FUNCTION_BLOCK EM_DockingInterface EXTENDS EM_Base
VAR CONSTANT 
	c_nResultDataSize : UINT := 20;
END_VAR
VAR
//------------------------------------------//
//Control Modules (Devices)
	cmValveDockingClampsUpper : CM_ValveWithDoubleFB;
	cmValveDockingClampsLower : CM_ValveWithDoubleFB;
	cmValveUnlockingPinsUpper : CM_ValveWithFB;
	cmValveUnlockingPinsLower : CM_ValveWithFB;
	
//------------------------------------------//

//------------------------------------------//
//Inputs
		s_diStaBoxAtPreDockingPosition : FB_DigInput;
		s_diStaSensorBoxAtDockedPosition : FB_DigInput;
		
//------------------------------------------//
	
//------------------------------------------//
//Outputs

//------------------------------------------//


//Requests
	s_bReqDockBox : BOOL := FALSE;
	s_bReqUndockBox : BOOL := FALSE;
	
//Properties
	s_bStaDockingDone : BOOL := FALSE;
	s_bStaUndockingDone : BOOL := FALSE;
	
	
//Alarms

//Warnings
	fbAlarmHandlerNoBoxPresentAtPreDockingPosition : FB_AlarmHandler;
	fbAlarmHandlerNoBoxPresentAtDockedPosition : FB_AlarmHandler;

	s_bWrnNoBoxPresentAtPreDockingPosition : BOOL;
	s_bWrnNoBoxPresentAtDockedPosition : BOOL;
	
//------------------------------------------//
//Params
	//Tool settings
	s_fbParamToolHardwareNr				: FB_HmiParamHandler;
    s_fbParamToolSoftwareVersion		: FB_HmiParamHandler;

	s_fbParamName						: FB_HmiParamHandler;
	s_fbParamNumber						: FB_HmiParamHandler;
	s_fbParamRevision                   : FB_HmiParamHandler;
	
	s_fbParamTeslaMeterIp				: FB_HmiParamHandler;
	s_fbParamTeslaMeterPort				: FB_HmiParamHandler;
	
	//Product settings (Maybe)
	s_fbParamTotalStroke				: FB_HmiParamHandler;
	s_fbParamStepStroke					: FB_HmiParamHandler;
	s_fbParamAveragingNumberTest		: FB_HmiParamHandler;
	
	s_fbParamaMaxMagnitudeCriteria		: FB_HmiParamHandler;
	
	s_fbParamRefIduBottom				: FB_HmiParamHandler;
	s_fbParamRefItm                     : FB_HmiParamHandler;
	s_fbParamRefCenterTpmPipe           : FB_HmiParamHandler;
	s_fbParamRefCpValve					: FB_HmiParamHandler;
//------------------------------------------//

//------------------------------------------//
//Variables
	s_sTestResult 						: STRING;
	
	s_eSeqDockingInterface : E_SeqDockingInterface;
	s_fbSeqDockingInterface : FB_SeqControl;
	
	s_eCurrentTest						: E_TestMode;
//--	s_stCommandsTesla					: ST_SCPI_TeslaCommands;
	
	
	// Interlocks
	s_bIlckSpeedDoorOuterToOpen 		: BOOL := TRUE;
	s_bIlckSpeedDoorOuterToClose 		: BOOL := TRUE;
	
	s_bIlckDoorLockCleanroomToOpen 		: BOOL := TRUE;
	
//------------------------------------------//

//------------------------------------------//
//Sensor data	
	s_aMagneticX						: ARRAY[0..c_nResultDataSize] OF LREAL;
	s_aMagneticY						: ARRAY[0..c_nResultDataSize] OF LREAL;
	s_aMagneticZ						: ARRAY[0..c_nResultDataSize] OF LREAL;
	s_aMagneticMagnitude				: ARRAY[0..c_nResultDataSize] OF LREAL;
	s_aProbePositionZ					: ARRAY[0..c_nResultDataSize] OF LREAL;
	
	s_sXMLData							: STRING(Param_Project.n_MaxLenghtXmlDbRow*Param_Project.n_NumberofRowsXmlDb);
	
	s_aHmi_MagneticTest					: ARRAY[1..3,0..c_nResultDataSize] OF ST_POINT;
	
//	s_aHmi_ProbePositionZ				: ARRAY[1..1,1..GVL_Datalogging.c_nHmiLogSize] OF ST_POINT;
//------------------------------------------//

//------------------------------------------//
//Alarms

//------------------------------------------//

//------------------------------------------//
//Hmi
	s_nToHmiStepNr						: INT;
	s_nToHmiMaxStepNr					: INT;
	s_sToHmiInstructionText				: T_MAXSTRING;
	s_sToHmiProcedure					: T_MAXSTRING;
	
	s_fbHmiBtnStart						: FB_HmiBtn;
	s_fbHmiBtnStop						: FB_HmiBtn;	
	s_fbHmiBtnDiagnosticsLogging		: FB_HmiBtn;
	
	s_fbHmiProbeMotor 					: Hmi_Motor_Base;
	
	s_fbHmiBtnEnableMotor				: FB_HmiBtn;
	s_fbHmiBtnHomeMotor					: FB_HmiBtn;
	s_fbHmiBtnGetField					: FB_HmiBtn;
	
	s_fbHmiLedHomedMotor				: FB_HmiLed;
	s_fbHmiTableDownPressed				: FB_HmiLed;
	s_fbHmiStopPressed					: FB_HmiLed;
	s_fbHmiTableDownSensor				: FB_HmiLed;
//------------------------------------------//
END_VAR


SUPER^();

METHOD PROTECTED _m_Alarms : BOOL





IF NOT SUPER^._m_Alarms() THEN
	RETURN;
END_IF

// Set error bits

// Alarm Handlers
fbAlarmHandlerNoBoxPresentAtPreDockingPosition(
	i_bStaActive := s_bWrnNoBoxPresentAtPreDockingPosition, 
	i_eAlarmLevel := E_AlarmLevel.Warning, 
	i_sAlarmText := 'No box present at per-docking position');
	
fbAlarmHandlerNoBoxPresentAtDockedPosition(
	i_bStaActive := s_bWrnNoBoxPresentAtDockedPosition, 
	i_eAlarmLevel := E_AlarmLevel.Warning, 
	i_sAlarmText := 'No box present at docked position');

// Reset warnings
IF i_bCmdReset THEN
	s_bWrnNoBoxPresentAtPreDockingPosition := FALSE;
	s_bWrnNoBoxPresentAtDockedPosition := FALSE;
END_IF	
	
_m_Alarms := TRUE;
END_METHOD

METHOD PROTECTED _m_Devices : BOOL

IF NOT SUPER^._m_Devices() THEN
	RETURN;
END_IF


s_diStaBoxAtPreDockingPosition(
	i_stSettings := );

s_diStaSensorBoxAtDockedPosition(
	i_stSettings := );

cmValveDockingClampsUpper(
	i_bReqEnable := i_bReqEnable,
	i_eCtrlMode := i_eCtrlMode,
	i_bCmdReset := i_bCmdReset,
	i_sCmName := 'Docking clamps upper', 
	i_stSettings := );
	
cmValveDockingClampsLower(
	i_bReqEnable := i_bReqEnable,
	i_eCtrlMode := i_eCtrlMode,
	i_bCmdReset := i_bCmdReset,
	i_sCmName := 'Docking clamps lower',
	i_stSettings := );
	
cmValveUnlockingPinsUpper(
	i_bReqEnable := i_bReqEnable,
	i_eCtrlMode := i_eCtrlMode,
	i_bCmdReset := i_bCmdReset,
	i_sCmName := 'Unloacking pins upper',
	i_stSettings := );
	
cmValveUnlockingPinsLower(
	i_bReqEnable := i_bReqEnable,
	i_eCtrlMode := i_eCtrlMode,
	i_bCmdReset := i_bCmdReset,
	i_sCmName := 'Unloacking pins lower',
	i_stSettings := );
	
(*	
	// Interlocks (doors must work as an airlock, only one door may be opened at all times)
	s_bIlckSpeedDoorOuterToOpen :=
		s_cmDoorLockCleanroom.p_bStaError
		OR NOT(s_cmDoorLockCleanroom.p_bStaEnabled)
		NOT(s_cmDoorLockCleanroom.p_bStaDoorIsClosed)
		OR NOT (s_cmDoorLockCleanroom.p_bStaLockIsApplied)
		OR s_cmDoorLockCleanroom.p_bStaLockIsReleased
		OR TRUE (*Air treathment unit must be running and ok*)
		OR TRUE (*Add more..*);
	s_bIlckSpeedDoorOuterToClose :=
		TRUE (*Opening must be free*)
		OR TRUE (*Add more..*);
	
	s_bIlckDoorLockCleanroomToOpen :=
		s_cmSpeedDoorOuter.p_bStaError
		OR NOT(s_cmSpeedDoorOuter.p_bStaEnabled)
		OR NOT(s_cmSpeedDoorOuter.p_bStaIsClosed)
		OR s_cmSpeedDoorOuter.p_bStaIsClosing
		OR s_cmSpeedDoorOuter.p_bStaIsOpened
		OR s_cmSpeedDoorOuter.p_bStaIsOpening
		OR TRUE (*Air treathment unit must be running and ok*)
		OR TRUE (*Add more..*);
*)	
_m_Devices := TRUE;
END_METHOD

METHOD PROTECTED _m_Hmi : BOOL

IF NOT SUPER^._m_Hmi() THEN
	RETURN;
END_IF

s_fbHmiBtnDiagnosticsLogging();
s_fbHmiBtnStart();
s_fbHmiBtnStop();

s_fbHmiBtnEnableMotor();
s_fbHmiBtnHomeMotor();
s_fbHmiBtnGetField();

s_fbHmiProbeMotor(i_IMotor := s_CmProbeMotor);

s_fbHmiLedHomedMotor(i_bStaLed := s_CmProbeMotor.p_bStaMotorHomed);
s_fbHmiTableDownPressed(i_bStaLed := s_diBtnTableDown.p_bStaInput);
s_fbHmiTableDownSensor(i_bStaLed := s_diTableDownSensor.p_bStaInput);
s_fbHmiStopPressed(i_bStaLed := s_diBtnStop.p_bStaInput);

_m_Hmi := TRUE;
END_METHOD

METHOD PROTECTED _m_Init : BOOL

IF NOT SUPER^._m_Init() THEN
	RETURN;
END_IF

//----------------------------------//
//CM
	s_cmSpeedDoorOuter.i_stSettings.

	s_CmProbeMotor.i_bReqEnable						:= FALSE;
	s_CmProbeMotor.i_sCmName 						:= 'Probe motor';
	s_CmProbeMotor.i_eBtnCtrlType					:= E_HmiButtonType.PUSHBUTTON;
	s_CmProbeMotor.i_bCfgReverseDirection			:= FALSE;
	s_CmProbeMotor.p_bCfgMovingForward				:= TRUE;
	s_CmProbeMotor.p_bCfgMovingReverse				:= TRUE;
	s_CmProbeMotor.p_fSetMotorVelo					:= 10;
	
	s_CmProbeMotor.i_stSettings.i_fAccelaration 	:= 1000;
	s_CmProbeMotor.i_stSettings.i_fDecelaration		:= 1000;
	s_CmProbeMotor.i_stSettings.i_fJerk				:= 10000;
	
	s_CmTeslaMeter.i_bReqEnable						:= FALSE;
	s_CmTeslaMeter.i_stSettings.tConnectionTimeOut	:= T#5S;

	
//---------------------------------//	
	
//----------------------------------//	
//Hmi 
	s_fbHmiBtnDiagnosticsLogging.p_eButtontype 			:= E_HmiButtonType.TOGGLEBUTTON;
	s_fbHmiBtnDiagnosticsLogging.p_bStaVisible 			:= TRUE;
	s_fbHmiBtnDiagnosticsLogging.p_bStaEnabled 			:= TRUE;
	s_fbHmiBtnDiagnosticsLogging.p_sBtnText				:= 'Diagnostics Logging';
	
	s_fbHmiBtnStart.p_eButtontype 						:= E_HmiButtonType.PUSHBUTTON;
	s_fbHmiBtnStart.p_bStaVisible 						:= FALSE;
	s_fbHmiBtnStart.p_bStaEnabled 						:= FALSE;		
	s_fbHmiBtnStart.p_sBtnText							:= 'Start';

	s_fbHmiBtnStop.p_eButtontype 						:= E_HmiButtonType.PUSHBUTTON;
	s_fbHmiBtnStop.p_bStaVisible 						:= FALSE;
	s_fbHmiBtnStop.p_bStaEnabled 						:= FALSE;		
	s_fbHmiBtnStop.p_sBtnText							:= 'Stop';
	
	s_fbHmiBtnEnableMotor.p_eButtontype 				:= E_HmiButtonType.TOGGLEBUTTON;
	s_fbHmiBtnEnableMotor.p_bStaVisible 				:= TRUE;
	s_fbHmiBtnEnableMotor.p_bStaEnabled 				:= FALSE;		
	s_fbHmiBtnEnableMotor.p_sBtnText					:= 'Enable motor';
	
	s_fbHmiBtnGetField.p_eButtontype 					:= E_HmiButtonType.PUSHBUTTON;
	s_fbHmiBtnGetField.p_bStaVisible 					:= TRUE;
	s_fbHmiBtnGetField.p_bStaEnabled 					:= FALSE;		
	s_fbHmiBtnGetField.p_sBtnText						:= 'Get magnetic field';
	
	s_fbHmiBtnHomeMotor.p_eButtontype 					:= E_HmiButtonType.PUSHBUTTON;
	s_fbHmiBtnHomeMotor.p_bStaVisible 					:= TRUE;
	s_fbHmiBtnHomeMotor.p_bStaEnabled 					:= FALSE;		
	s_fbHmiBtnHomeMotor.p_sBtnText						:= 'Home motor';
//----------------------------------//	


//----------------------------------//	
//Initialize all moving averages

//----------------------------------//	

//----------------------------------//	
//Inputs
s_diTableDownSensor.i_stSettings.tmInputDelay	:= T#0S;	
s_diBtnTableDown.i_stSettings.tmInputDelay		:= T#0S;
s_diBtnStop.i_stSettings.tmInputDelay			:= T#0S;
//----------------------------------//	

//----------------------------------//	
//Inputs
s_doRelayTableDown.i_stSettings.bCfgDelay		:= FALSE;	
s_doRelayTableDown.i_stSettings.tmOutputDelay	:= T#0S;	
//----------------------------------//	

_m_Init := TRUE;
END_METHOD

METHOD PROTECTED _m_Inputs : BOOL

IF NOT SUPER^._m_Inputs() THEN
	RETURN;
END_IF

s_diStaBoxAtPreDockingPosition();
s_diStaSensorBoxAtDockedPosition();

_m_Inputs := TRUE;
END_METHOD

METHOD PROTECTED _m_Outputs : BOOL

IF NOT SUPER^._m_Outputs() THEN
	RETURN;
END_IF

s_doRelayTableDown(); //i_bStaOutput written in procedure or manual mode

_m_Outputs := TRUE;
END_METHOD

METHOD PROTECTED _m_Params : BOOL
VAR_INST
	s_fToHmiXAxisMin	: LREAL;
	s_fToHmiXAxisMax	: LREAL;
	s_fToHmiYAxisMin	: LREAL;
	s_fToHmiYAxisMax	: LREAL;
END_VAR

IF NOT SUPER^._m_Params() THEN
	RETURN;
END_IF

s_fbParamToolHardwareNr(i_fDefaultValue				:= 0,
						i_nArrayFolderIndex			:= 1,
						i_sName						:= 'Harware ID',
						i_bIsNumber					:= FALSE);

s_fbParamToolSoftwareVersion(i_fDefaultValue		:= 0,
							i_nArrayFolderIndex		:= 1,
							i_sName					:= 'Software Version',
							i_bIsNumber				:= FALSE);

s_fbParamName(i_fDefaultValue						:= 0,
				i_nArrayFolderIndex					:= 1,
				i_sName								:= 'Description',
				i_bIsNumber							:= FALSE);
							
s_fbParamTeslaMeterIp(i_fDefaultValue			:= 0,
						i_nArrayFolderIndex		:= 1,
						i_sName					:= 'Tesla meter ip adress',
						i_bIsNumber				:= FALSE);
						
s_fbParamTeslaMeterPort(i_fDefaultValue			:= 0,
						i_nArrayFolderIndex		:= 1,
						i_sName					:= 'Tesla meter port number',
						i_bIsNumber				:= TRUE);

//---------

						
s_fbParamTotalStroke(i_fDefaultValue			:= 100,
						i_nArrayFolderIndex		:= 2,
						i_sName					:= 'Total measurement stroke',
						i_bIsNumber				:= TRUE);
						
s_fbParamStepStroke(i_fDefaultValue				:= 10,
						i_nArrayFolderIndex		:= 2,
						i_sName					:= 'Step distance per measurement',
						i_bIsNumber				:= TRUE);

s_fbParamAveragingNumberTest(i_fDefaultValue		:= 10,
							i_nArrayFolderIndex		:= 2,
							i_sName					:= 'Number of measurements per step for averaging the magnetic field',
							i_bIsNumber				:= TRUE);
							
s_fbParamaMaxMagnitudeCriteria(i_fDefaultValue		:= 100,
							i_nArrayFolderIndex		:= 2,
							i_sName					:= 'Maximum allowed magnitude magnetic field (Test)',
							i_bIsNumber				:= TRUE);

s_fbParamRefIduBottom(i_fDefaultValue				:= 0,
							i_nArrayFolderIndex		:= 2,
							i_sName					:= 'Distance from home position to lower IDU Bottom',
							i_bIsNumber				:= TRUE);
							
s_fbParamRefItm(i_fDefaultValue						:= 0,
							i_nArrayFolderIndex		:= 2,
							i_sName					:= 'Distance from home position Itm lower IDU / upper IDU',
							i_bIsNumber				:= TRUE);
							
s_fbParamRefCenterTpmPipe(i_fDefaultValue			:= 0,
							i_nArrayFolderIndex		:= 2,
							i_sName					:= 'Distance from home position to centre TPM pipe',
							i_bIsNumber				:= TRUE);
							
s_fbParamRefCpValve(i_fDefaultValue		:= 0,
							i_nArrayFolderIndex		:= 2,
							i_sName					:= 'Distance from home position to bottom C/P valve',
							i_bIsNumber				:= TRUE);				

GVL_DataLogging.g_stReportData.CabinetSerialNumber      := s_fbParamToolHardwareNr.p_sValue;
GVL_DataLogging.g_stReportData.TesterSoftwareVersion    := s_fbParamToolSoftwareVersion.p_sValue;
GVL_DataLogging.g_stReportData.Operator                 := GVL.g_sUser;
GVL_DataLogging.g_stReportData.Note						:= GVL.g_sNotesEntry;
//GVL_DataLogging.g_stReportData.Message can be filled in test procedure with for example the error if test is stopped
GVL_DataLogging.g_stReportData.SerialNumber             := GVL.g_sSerialNumber;

s_fToHmiXAxisMin	:= -2*s_fbParamaMaxMagnitudeCriteria.p_fValue;
s_fToHmiXAxisMax	:= 2*s_fbParamaMaxMagnitudeCriteria.p_fValue;
s_fToHmiYAxisMin	:= s_CmProbeMotor.p_fHomePosition;
s_fToHmiYAxisMax	:= s_fbParamRefCpValve.p_fValue*1.2;

_m_Params := TRUE;
END_METHOD

METHOD PUBLIC m_DockBox : BOOL

s_bReqDockBox := TRUE;
s_bReqUndockBox := FALSE;

m_DockBox := TRUE;
END_METHOD

METHOD PUBLIC m_Main : BOOL

IF NOT SUPER^.m_Main() THEN
	RETURN;
END_IF


CASE i_eCtrlMode OF

	E_CtrlMode.IDLE:
		;
		
	E_CtrlMode.AUTOMATIC:
		
		s_fbSeqDockingInterface(
			i_nSeqStep := s_eSeqDockingInterface, 
			i_sStepName := , 
			i_bCmdReset := i_bCmdReset, 
			i_bStaError := s_bStaError, 
			q_bStaEntry => , 
			q_tmStepTime => , 
			q_eActState => );
	
		CASE s_eSeqDockingInterface OF
			
			E_SeqDockingInterface.IDLE:
			
				IF s_bReqDockBox THEN
					IF s_diStaBoxAtPreDockingPosition.p_bStaInputDelayed THEN
						s_eSeqDockingInterface := E_SeqDockingInterface.DOCKING_CLOSE_CLAMPS;
					ELSE
						s_bWrnNoBoxPresentAtPreDockingPosition := TRUE;	
					END_IF
				END_IF
				
				IF s_bReqUndockBox THEN
					IF s_diStaSensorBoxAtDockedPosition.p_bStaInputDelayed THEN
						s_eSeqDockingInterface := E_SeqDockingInterface.UNDOCKING_LOCK_DOOR;
					ELSE
						s_bWrnNoBoxPresentAtDockedPosition := TRUE;	
					END_IF	
					
				END_IF
			
				IF s_bReqDockBox AND s_diStaBoxAtPreDockingPosition.p_bStaInputDelayed THEN
					s_eSeqDockingInterface := E_SeqDockingInterface.DOCKING_CLOSE_CLAMPS; 
				ELSIF s_bReqUndockBox THEN	
					s_eSeqDockingInterface := E_SeqDockingInterface.UNDOCKING_LOCK_DOOR;
				END_IF
				
			E_SeqDockingInterface.DOCKING_CLOSE_CLAMPS:
				
				IF s_fbSeqDockingInterface.q_bStaEntry THEN 
					cmValveDockingClampsUpper.m_On();
					cmValveDockingClampsLower.m_On();
				END_IF
				
				IF cmValveDockingClampsUpper.p_bStaIsOn AND cmValveDockingClampsLower.p_bStaIsOn THEN
					s_eSeqDockingInterface := E_SeqDockingInterface.DOCKING_UNLOCK_DOOR;
				ELSIF cmValveDockingClampsUpper.p_bStaError OR cmValveDockingClampsLower.p_bStaError THEN 
					s_eSeqDockingInterface := E_SeqDockingInterface.ERROR;
					// write down some info?
				ELSIF s_fbSeqDockingInterface.q_tmStepTime >= T#30S THEN
 					s_eSeqDockingInterface := E_SeqDockingInterface.ERROR;
					// write down some info?
				END_IF
			
			E_SeqDockingInterface.DOCKING_UNLOCK_DOOR:
			
				IF s_fbSeqDockingInterface.q_bStaEntry THEN 
					cmValveUnlockingPinsUpper.m_On();
					cmValveUnlockingPinsLower.m_On();
				END_IF
				
				IF cmValveUnlockingPinsUpper.p_bStaIsOn AND cmValveUnlockingPinsLower.p_bStaIsOn THEN
					s_eSeqDockingInterface := E_SeqDockingInterface.DOCKING_DONE;
				ELSIF cmValveUnlockingPinsUpper.p_bStaError OR cmValveUnlockingPinsLower.p_bStaError THEN 
					s_eSeqDockingInterface := E_SeqDockingInterface.ERROR;
					// write down some info?
				ELSIF s_fbSeqDockingInterface.q_tmStepTime >= T#30S THEN
 					s_eSeqDockingInterface := E_SeqDockingInterface.ERROR;
					// write down some info?
				END_IF
			
			E_SeqDockingInterface.DOCKING_DONE:
				s_eSeqDockingInterface := E_SeqDockingInterface.IDLE;
			
			E_SeqDockingInterface.UNDOCKING_LOCK_DOOR:
			
				IF s_fbSeqDockingInterface.q_bStaEntry THEN 
					cmValveUnlockingPinsUpper.m_Off();
					cmValveUnlockingPinsLower.m_Off();
				END_IF
				
				IF cmValveUnlockingPinsUpper.p_bStaIsOff AND cmValveUnlockingPinsLower.p_bStaIsOff THEN
					s_eSeqDockingInterface := E_SeqDockingInterface.UNDOCKING_OPEN_CLAMPS;
				ELSIF cmValveUnlockingPinsUpper.p_bStaError OR cmValveUnlockingPinsLower.p_bStaError THEN 
					s_eSeqDockingInterface := E_SeqDockingInterface.ERROR;
					// write down some info?
				ELSIF s_fbSeqDockingInterface.q_tmStepTime >= T#30S THEN
 					s_eSeqDockingInterface := E_SeqDockingInterface.ERROR;
					// write down some info?
				END_IF
				
			E_SeqDockingInterface.UNDOCKING_OPEN_CLAMPS:
			
				IF s_fbSeqDockingInterface.q_bStaEntry THEN 
					cmValveDockingClampsUpper.m_Off();
					cmValveDockingClampsLower.m_Off();
				END_IF
				
				IF cmValveDockingClampsUpper.p_bStaIsOff AND cmValveDockingClampsLower.p_bStaIsOff THEN
					s_eSeqDockingInterface := E_SeqDockingInterface.UNDOCKING_DONE;
				ELSIF cmValveDockingClampsUpper.p_bStaError OR cmValveDockingClampsLower.p_bStaError THEN 
					s_eSeqDockingInterface := E_SeqDockingInterface.ERROR;
					// write down some info?
				ELSIF s_fbSeqDockingInterface.q_tmStepTime >= T#30S THEN
 					s_eSeqDockingInterface := E_SeqDockingInterface.ERROR;
					// write down some info?
				END_IF
				
			E_SeqDockingInterface.UNDOCKING_DONE:
				s_eSeqDockingInterface := E_SeqDockingInterface.IDLE;
				
			E_SeqDockingInterface.READY:
				;
			
			E_SeqDockingInterface.ERROR:
				
				IF i_bCmdReset THEN
					//Reset errors (probebly alredy done in the methode devices)
					//--cmValveDockingClampsUpper.i_bCmdReset := TRUE;
				
					s_eSeqDockingInterface := E_SeqDockingInterface.IDLE;
				END_IF
				
		END_CASE		
	
		
	E_CtrlMode.MANUAL:
		;
	

END_CASE

//-- Old code as an example
(*
CASE i_eCtrlMode OF
	E_CtrlMode.IDLE:
		IF s_CmProbeMotor.p_bStaEnabled THEN
			s_CmProbeMotor.m_DisableAxis();
			s_fbHmiBtnEnableMotor.m_Off();
			s_fbHmiBtnHomeMotor.p_bStaEnabled := FALSE;
		END_IF
		
		s_eCurrentTest	:= 	E_TestMode.IDLE;
	
		s_fbHmiBtnStop.p_bStaVisible := FALSE;
		s_fbHmiBtnStop.p_bStaEnabled := FALSE;		
		
	E_CtrlMode.AUTOMATIC:
		
		CASE s_eCurrentTest OF
			E_TestMode.IDLE:
				GVL.g_bLedFlashSlow			:= FALSE;
				
				s_CmProbeMotor.i_bReqEnable	:= FALSE;
			
				GVL_KMWEGenericLib.g_fbHmiBtnReturn.p_bStaEnabled 	:= TRUE;
				GVL_KMWEGenericLib.g_fbHmiBtnReturn.p_bStaVisible 	:= TRUE;
				
				IF GVL.g_sToHmiMiddleContent = GVL.g_stHmiMiddle.OperatorInputData THEN
					IF NOT GVL_KMWEGenericLib.g_fbAlarmManager.p_bAlarmActive THEN
						s_fbHmiBtnStart.p_bStaVisible	:= TRUE;
						s_fbHmiBtnStart.p_bStaEnabled	:= TRUE;
					ELSE
						s_fbHmiBtnStart.p_bStaVisible	:= FALSE;
						s_fbHmiBtnStart.p_bStaEnabled	:= FALSE;
					END_IF
				END_IF
				
				IF s_fbHmiBtnStart.p_osrBtnPress THEN
					s_eCurrentTest := E_TestMode.Magnetic; 
				END_IF 
				
			E_TestMode.Magnetic:	
				_m_Procedure_Test(i_bCmdReset			:= s_fbHmiBtnStart.p_osfBtnPress, 
									i_bStaError			:= GVL_KMWEGenericLib.g_fbAlarmManager.p_bAlarmActive OR s_fbHmiBtnStop.p_osrBtnPress OR s_diBtnStop.p_osrOn);
		END_CASE
		
	E_CtrlMode.MANUAL:
		_m_Manual(i_bCmdReset			:= GVL.g_UnRMMT.s_fbHmiBtnManual.p_osfBtnPress OR GVL_KMWEGenericLib.g_fbAlarmManager.p_osrReset, 
					i_bStaError			:= GVL_KMWEGenericLib.g_fbAlarmManager.p_bAlarmActive OR s_fbHmiBtnStop.p_osrBtnPress OR s_diBtnStop.p_osrOn);	
END_CASE
*)
END_METHOD

METHOD PUBLIC m_UndockBox : BOOL






s_bReqDockBox := FALSE;
s_bReqUndockBox := TRUE;

m_UndockBox := TRUE;
END_METHOD

PROPERTY PUBLIC p_bStaDockingDone : BOOL
GET

p_bStaDockingDone := s_bStaDockingDone;
END_GET
END_PROPERTY

PROPERTY p_bStaUndockingDone : BOOL
GET

p_bStaUndockingDone := s_bStaUndockingDone;
END_GET
END_PROPERTY

END_FUNCTION_BLOCK

(* stored: Version 1.1.0.1, ProductVersion 3.1.4024.12
   POU EM_DockingInterface: Id {1a98308c-f0e0-4a53-963d-dfa6a727e4cb}, SpecialFunc None
   Method _m_Alarms: Id {c0cf83f3-e704-4016-bd6f-2d30156087ff}
   Method _m_Devices: Id {b43c077f-3abc-4642-868d-7667cd19393f}
   Method _m_Hmi: Id {5090ba0a-8e2b-4ba6-88b3-b451c7c7863d}
   Method _m_Init: Id {f248bb7d-4543-4fa5-93e5-377095a1130a}
   Method _m_Inputs: Id {15e5d91e-088b-4383-82aa-ad9257b81a9b}
   Method _m_Outputs: Id {748b7abf-6524-428b-ad1f-dd34bf2d901c}
   Method _m_Params: Id {78648659-4a86-4875-84af-aa8b2b68e067}
   Method m_DockBox: Id {8e382bf6-1d32-4474-a8a5-7c183a3c7036}
   Method m_Main: Id {13829dfc-fc98-4f3a-8520-8dee66cb84d9}
   Method m_UndockBox: Id {b328f671-5464-49bf-836c-f1f93f3d32af}
   Property p_bStaDockingDone: Id {a61394df-c5f0-450a-8cdf-e47379cb8b81}
   Get Get: Id {e6843217-13bc-4765-b8f6-a237563e9d39}
   Property p_bStaUndockingDone: Id {bb261a88-cc34-4fd6-bf54-1089f44f9408}
   Get Get: Id {44b7df0c-94a7-4b6d-a3a8-e5b8bd6f931a} *)
